PROGRAM ST10_BarcodeScanner
VAR
	fbCognexBarcodeScanner: FB_CognexBarcodeScanner;
END_VAR

fbCognexBarcodeScanner(
	In_bManualMode:= G_MachineControl.stMachineOperateMode.MANUAL,
	In_bAutoMode:= G_MachineControl.stMachineOperateMode.AUTO OR G_MachineControl.stMachineOperateMode.DRYRUN,
	In_timeScanTimer:= T#10S, 
	In_iResultByte:= 20, 
	In_ioDeviceFault := G_Scanner.In_Signal_Conveyor.In_GeneralFault,
	In_ioTriggerReady:= G_Scanner.In_Signal_Conveyor.In_TriggerReady, 
	In_ioTriggerAck:= G_Scanner.In_Signal_Conveyor.In_TriggerAck, 
	In_ioAcquiring:= G_Scanner.In_Signal_Conveyor.In_Acquiring, 
	In_ioArrayData:= G_Scanner.In_Signal_Conveyor.In_ResultData, 
	Out_bDeviceError=> G_Error.E10_BarcodeScannerDeviceError,
	Out_bErrScanTimeOut=> G_Error.E10_BarcodeTimeout, 
	Out_ioTriggerEnable=> G_Scanner.Out_Signal_Conveyor.Out_TriggerEnable, 
	Out_ioTrigger=> G_Scanner.Out_Signal_Conveyor.Out_Trigger, 
	Out_bEnableReady=> G_Manual.M10_bTriggerScannerEnableReady,
	Out_bEnableReady=> G_Auto.A10_bTriggerScannerEnableReady,
	Out_bTriggerDone=> G_Manual.M10_bTriggerScannerDone,
	Out_bTriggerDone=> G_Auto.A10_bTriggerScannerDone,
	Out_sAutoBarcode=> G_Auto.A10_sScannerBarcode, 
	Out_sManualBarcode=> G_Manual.M10_sScannerBarcode, 
	Out_GetBarcodeDone=> G_Auto.A10_bScannerResultDone,
	Out_GetBarcodeDone=> G_Manual.M10_bScannerResultDone, 
	InOut_bAutoTriggerEnable:= G_Auto.A10_bTriggerScannerEnable, 
	InOut_bManualTriggerEnable:= G_Manual.M10_bTriggerScannerEnable, 
	InOut_bAutoTrigger:= G_Auto.A10_bTriggerScanner,
	InOut_bManualTrigger:= G_Manual.M10_bTriggerScanner);

END_PROGRAM

(* stored: Version 1.1.0.1, ProductVersion 3.1.4024.11
   POU ST10_BarcodeScanner: Id {c1db312c-c80d-4816-831f-8a2d1d2e41b9}, SpecialFunc None *)
